# EPICS autosave request: iocs/pvaDriverIOC/iocBoot/iocPvaDriver/auto_settings.req
file "NDStdArrays_settings.req",    P=$(P),  R=image1:
file "commonPlugin_settings.req",   P=$(P)
